GLOBALCONSTANTS FIELDBUS_SIGNAL (* Certain Constants especially for valid, error and not available *)
  (* Standard: SAE J1939; ISO 11783; Description: Copyright (c) 2023 HR Agrartechnik GmbH This program and the accompanying materials are made available under the terms of the Eclipse Public License 2.0 which is available at https://www.eclipse.org/legal/epl-2.0/ SPDX-License-Identifier: EPL-2.0 *)
  (* Version 3.0, 2025-04-14, Patrick Aigner, changed package *)
  (* Version 1.0, 2023-06-06, Franz Höpfinger, HR Agrartechnik GmbH *)
  PACKAGE eclipse4diac::signalprocessing;
  VAR_GLOBAL CONSTANT
    REVERSE : BYTE := BYTE#16#0; (* Direction reverse *)
    DISABLED : BYTE := BYTE#16#0; (* Not enabled *)
    DISENGAGED : BYTE := BYTE#16#0; (* Switched off *)
    FORWARD : BYTE := BYTE#16#1; (* Direction forward *)
    ENABLED : BYTE := BYTE#16#1; (* Enabled *)
    ENGAGED : BYTE := BYTE#16#1; (* Switched on *)
    ERROR_INDI_2Bit : BYTE := BYTE#16#2; (* 2 bit error indicator *)
    NOT_AVAILABLE_2Bit : BYTE := BYTE#16#3; (* 2 bit not available *)
    DONT_CARE_2bit : BYTE := BYTE#16#3; (* 2 bit dont care *)
    ERROR_INDI_3Bit : BYTE := BYTE#16#6; (* 3 bit error indicator *)
    NOT_AVAILABLE_3Bit : BYTE := BYTE#16#7; (* 3 bit not available *)
    DONT_CARE_3bit : BYTE := BYTE#16#7; (* 3 bit dont care *)
    ERROR_INDI_4bit : BYTE := BYTE#16#E; (* 4 bit error indicator *)
    NOT_AVAILABLE_4bit : BYTE := BYTE#16#F; (* 4 bit not available *)
    DONT_CARE_4bit : BYTE := BYTE#16#F; (* 4 bit dont care *)
    VALID_SIGNAL_B : BYTE := BYTE#16#FA; (* 8 bit max value of valid signal *)
    ERROR_INDI_B : BYTE := BYTE#16#FE; (* 8 bit error indicator *)
    NOT_AVAILABLE_B : BYTE := BYTE#16#FF; (* 8 bit not available *)
    DONT_CARE_B : BYTE := BYTE#16#FF; (* 8 bit dont care *)
    VALID_SIGNAL_W : WORD := WORD#16#FAFF; (* 16 bit max value of valid signal *)
    ERROR_INDI_W : WORD := WORD#16#FE00; (* 16 bit error indicator min *)
    NOT_AVAILABLE_W : WORD := WORD#16#FF00; (* 16 bit not available min *)
    ERROR_INDI_WM : WORD := WORD#16#FEFF; (* 16 bit error indicator max *)
    NOT_AVAILABLE_WM : WORD := WORD#16#FFFF; (* 16 bit not available max *)
    DONT_CARE_W : WORD := WORD#16#FFFF; (* 16 bit dont care *)
    VALID_SIGNAL_DW : DWORD := DWORD#16#FAFFFFFF; (* 32 bit max value of valid signal *)
    ERROR_INDI_DW : DWORD := DWORD#16#FE000000; (* 32 bit error indicator min *)
    NOT_AVAILABLE_DW : DWORD := DWORD#16#FF000000; (* 32 bit not available min *)
    ERROR_INDI_DWM : DWORD := DWORD#16#FEFFFFFF; (* 32 bit error indicator max *)
    NOT_AVAILABLE_DM : DWORD := DWORD#16#FFFFFFFF; (* 32 bit not available max *)
  END_VAR
END_GLOBALCONSTANTS
